FUNCTION proj32_TupleStruct_4: DINT
VAR_INPUT
    tuple: TupleStruct_4;
END_VAR


        proj32_TupleStruct_4 := tuple.field32;

END_FUNCTION

(* stored: ProductVersion 3.1.0.18, Version 1.1.0.1 *)
